FUNCTION_BLOCK ROBOT_BIT_TRL
VAR_INPUT
	ROBPOZ : INT; // Robot pozíció száma
	
END_VAR

VAR_OUTPUT
	POZ1 :BOOL; //Kimenet bit MSB
	POZ2 :BOOL; //Kimenet
	POZ3 :BOOL; //Kimenet
	
END_VAR
VAR
	
END_VAR

CASE ROBPOZ OF
0:
POZ1 := 0;
POZ2 := 0;
POZ3 :=0;

1:
POZ1 := 1;
POZ2 :=0;
POZ3 :=0;

2:
POZ1 :=0;
POZ2 :=1;
POZ3 :=0;

3:
POZ1 :=1;
POZ2 :=1;
POZ3 :=0;

4:
POZ1 :=0;
POZ2 :=0;
POZ3 :=1;

5:
POZ1 :=1;
POZ2 :=0;
POZ3 :=1;

6:
POZ1 :=0;
POZ2 :=1;
POZ3 :=1;

7:
POZ1 :=1;
POZ2 :=1;
POZ3 :=1;

END_CASE

END_FUNCTION_BLOCK

(* stored: Version 1.1.0.1, ProductVersion 3.1.4024.11
   POU ROBOT_BIT_TRL: Id {444280b1-f2b5-4491-bf24-e44eef5bce93}, SpecialFunc None *)
